% RSLogix 500 project lab 8 prelab.RSS, saved by version 8.40.00.08 %
PROJECT "UNTITLED"    % processor: MicroLogix 1000 %

PROGRAM FILES
  LAD 2 "MAIN_PROG"  11 rungs
  LAD 3 "USER_FAULT"  1 rungs
  LAD 4 "HSC_INT"  1 rungs
  LAD 5 "STI_INT"  1 rungs
  LAD 6, 7, 8, 9, 10, 11, 12, 13, 14, 15, 16: only END

DATA FILES
  O0 OUTPUT  1 elements
  I1 INPUT  2 elements
  S2 STATUS  33 elements
  B3 BINARY  32 elements
  T4 TIMER  40 elements
  C5 COUNTER  32 elements
  R6 CONTROL  16 elements
  N7 INTEGER  105 elements

LADDER 2 "MAIN_PROG"
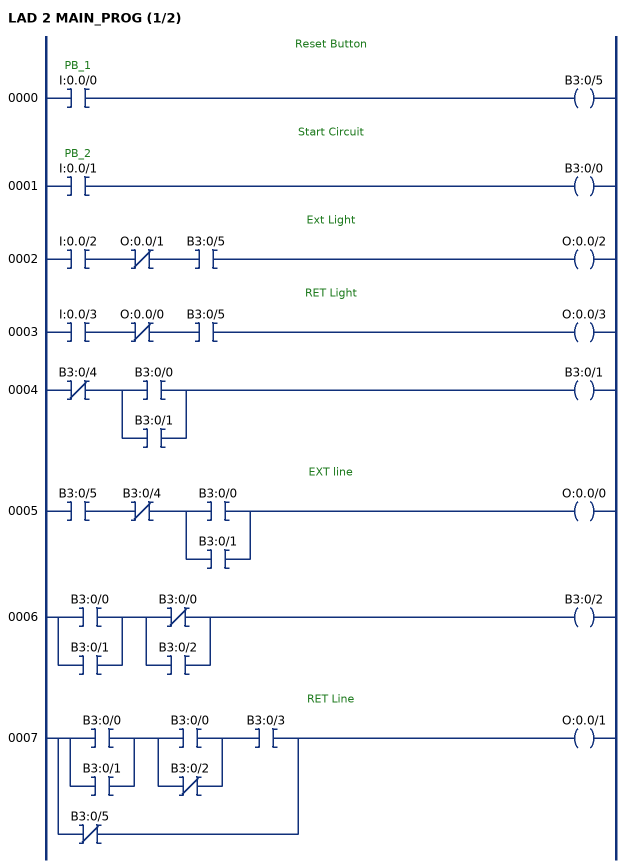
% Rung: 0 %
% Reset Button %
SOR XIC I:0.0/0 OTE B3:0/5 EOR
%   I:0.0/0  "PB_1" %
% Rung: 1 %
% Start Circuit %
SOR XIC I:0.0/1 OTE B3:0/0 EOR
%   I:0.0/1  "PB_2" %
% Rung: 2 %
% Ext Light %
SOR XIC I:0.0/2 XIO O:0.0/1 XIC B3:0/5 OTE O:0.0/2 EOR
% Rung: 3 %
% RET Light %
SOR XIC I:0.0/3 XIO O:0.0/0 XIC B3:0/5 OTE O:0.0/3 EOR
% Rung: 4 %
SOR XIO B3:0/4 BST XIC B3:0/0 NXB XIC B3:0/1 BND OTE B3:0/1 EOR
% Rung: 5 %
% EXT line %
SOR XIC B3:0/5 XIO B3:0/4 BST XIC B3:0/0 NXB XIC B3:0/1 BND OTE O:0.0/0 EOR
% Rung: 6 %
SOR BST XIC B3:0/0 NXB XIC B3:0/1 BND BST XIO B3:0/0 NXB XIC B3:0/2 BND OTE B3:0/2 EOR
% Rung: 7 %
% RET Line %
SOR BST BST XIC B3:0/0 NXB XIC B3:0/1 BND BST XIC B3:0/0 NXB XIO B3:0/2 BND XIC B3:0/3 NXB XIO B3:0/5 BND OTE O:0.0/1 EOR

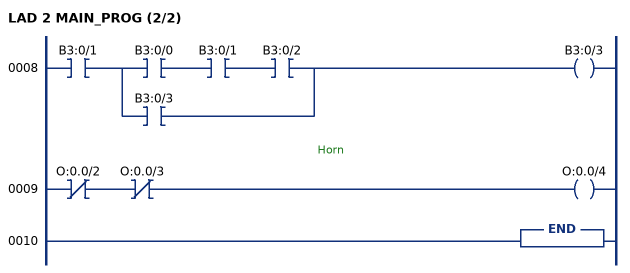
% Rung: 8 %
SOR XIC B3:0/1 BST XIC B3:0/0 XIC B3:0/1 XIC B3:0/2 NXB XIC B3:0/3 BND OTE B3:0/3 EOR
% Rung: 9 %
% Horn %
SOR XIO O:0.0/2 XIO O:0.0/3 OTE O:0.0/4 EOR
% Rung: 10 %
SOR END EOR
